FUNCTION_BLOCK AX_MERGE_2 (* Merge (OR) of two input events (generic FB) *)
  (* Standard: 61499-1 Annex A; Function: Output q is triggered when either SOCKET1 or SOCKET2 is received; Description: Copyright (c) 2026 HR Agrartechnik GmbH This program and the accompanying materials are made available under the terms of the Eclipse Public License 2.0 which is available at https://www.eclipse.org/legal/epl-2.0/ SPDX-License-Identifier: EPL-2.0 *)
  (* Version 3.0, 2026-01-14, Moritz Ortmeier, HR Agrartechnik GmbH *)
  PACKAGE adapter::events::unidirectional;
  IMPORT eclipse4diac::core::GenericClassName;
  IMPORT eclipse4diac::core::TypeHash;
  {SET_ATTRIBUTE(eclipse4diac::core::GenericClassName, 'GEN_E_MERGE')}
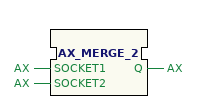
  SOCKETS
    SOCKET1 : adapter::types::unidirectional::AX; (* First input *)
    SOCKET2 : adapter::types::unidirectional::AX; (* Second input *)
  END_SOCKETS
  PLUGS
    Q : adapter::types::unidirectional::AX;
  END_PLUGS
END_FUNCTION_BLOCK
